TYPE CoolingRecycling :
STRUCT
	EN: BOOL := TRUE;
END_STRUCT
END_TYPE

(* stored: Version 1.1.0.1, ProductVersion 3.1.4024.6
   DUT CoolingRecycling: Id {0f58fd16-d1c7-48ff-9f22-ef910dfe5e29} *)
